# EPICS substitutions: CCD100/CCD100-IOC-01App/Db/unit_setter.substitutions
# Set points do not have units set because it will cause it to be processed thus sending a possibly wrong value
# to the display

file $(UTILITIES)/db/unit_setter.template {
  pattern
    {P,    FROM, TO}

    {"\$(P)", "UNITS", "READING"}
    {"\$(P)", "UNITS", "SP"}
	{"\$(P)", "UNITS", "SP:RBV"}
}
